PROGRAM P_ADS_ERR
VAR
	udiStationInError				: UDINT;
	udiStationErrorCode				: UDINT;
	sStationErrorDescription2		:WSTRING(255);

	
	fbRead_1: FB_ReadAdsSymByName;
	fbRead_2: FB_ReadAdsSymByName;
	fbRead_3: FB_ReadAdsSymByName;
	fbCyclicReadout: TON;
END_VAR

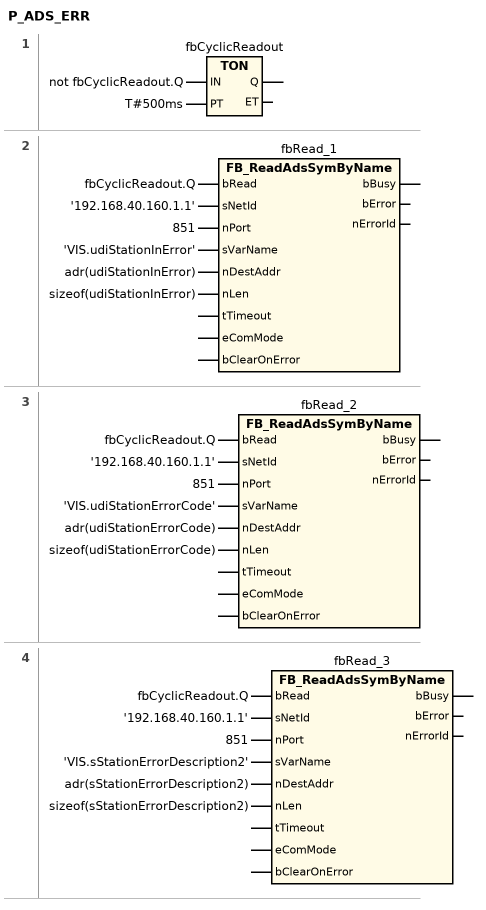
// NETWORK 1
fbCyclicReadout(IN := not fbCyclicReadout.Q, PT := T#500ms); // TON

// NETWORK 2
fbRead_1(
    bRead := fbCyclicReadout.Q,
    sNetId := '192.168.40.160.1.1',
    nPort := 851,
    sVarName := 'VIS.udiStationInError',
    nDestAddr := adr(udiStationInError),
    nLen := sizeof(udiStationInError)); // FB_ReadAdsSymByName

// NETWORK 3
fbRead_2(
    bRead := fbCyclicReadout.Q,
    sNetId := '192.168.40.160.1.1',
    nPort := 851,
    sVarName := 'VIS.udiStationErrorCode',
    nDestAddr := adr(udiStationErrorCode),
    nLen := sizeof(udiStationErrorCode)); // FB_ReadAdsSymByName

// NETWORK 4
fbRead_3(
    bRead := fbCyclicReadout.Q,
    sNetId := '192.168.40.160.1.1',
    nPort := 851,
    sVarName := 'VIS.sStationErrorDescription2',
    nDestAddr := adr(sStationErrorDescription2),
    nLen := sizeof(sStationErrorDescription2)); // FB_ReadAdsSymByName

END_PROGRAM

(* stored: Version 1.1.0.1, ProductVersion 3.1.4024.12
   POU P_ADS_ERR: Id {ca383858-8313-418a-8e8a-c2da2ce7bd4b}, SpecialFunc None *)
